// LS Electric XG5000 project: 과년71_1
// PLC NewPLC
// module base 0 slot 0: 입출력 모듈:XBC-DR20S (DC 24V 입력 12점, 릴레이 출력 8점)

PROGRAM NewProgram (task: 스캔 프로그램)

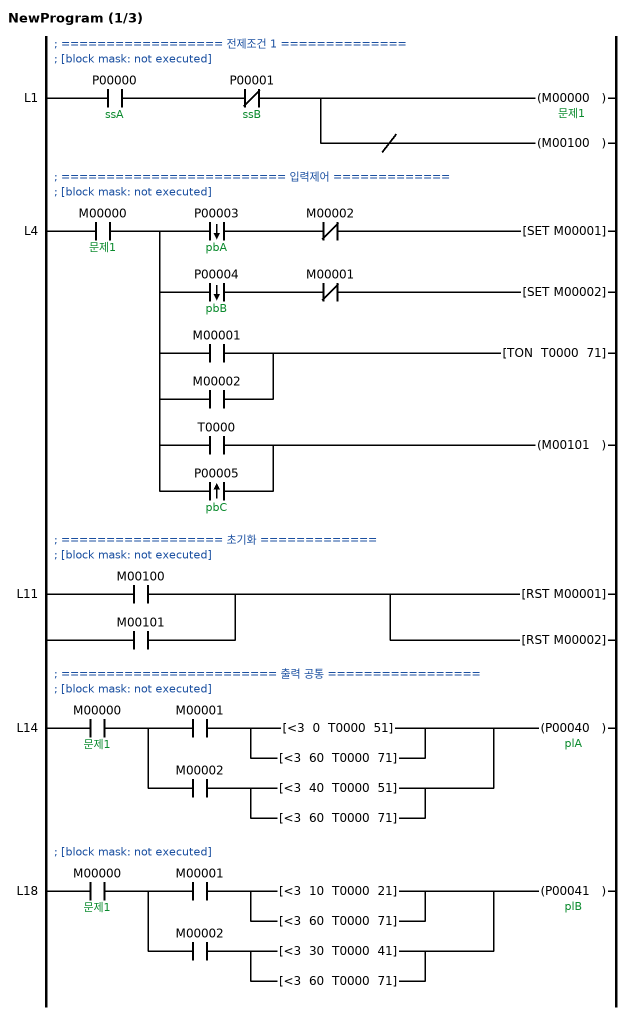
// ================== 전제조건 1 ==============
; L1 (block mask: not executed)
LOAD      P00000	// ssA
AND NOT   P00001	// ssB
OUT       M00000	// 문제1
NOT
OUT       M00100
// ========================= 입력제어 =============
; L4 (block mask: not executed)
LOAD      M00000	// 문제1
MPUSH
ANDN      P00003	// pbA
AND NOT   M00002
SET       M00001
MLOAD
ANDN      P00004	// pbB
AND NOT   M00001
SET       M00002
MLOAD
LOAD      M00001
OR        M00002
AND LOAD
TON       T0000 71
MPOP
LOAD      T0000
ORP       P00005	// pbC
AND LOAD
OUT       M00101
// ================== 초기화 =============
; L11 (block mask: not executed)
LOAD      M00100
OR        M00101
RST       M00001
RST       M00002
// ======================== 출력 공통 =================
; L14 (block mask: not executed)
LOAD      M00000	// 문제1
LOAD      M00001
LOAD<3    0 T0000 51
OR<3      60 T0000 71
AND LOAD
LOAD      M00002
LOAD<3    40 T0000 51
OR<3      60 T0000 71
AND LOAD
OR LOAD
AND LOAD
OUT       P00040	// plA
; L18 (block mask: not executed)
LOAD      M00000	// 문제1
LOAD      M00001
LOAD<3    10 T0000 21
OR<3      60 T0000 71
AND LOAD
LOAD      M00002
LOAD<3    30 T0000 41
OR<3      60 T0000 71
AND LOAD
OR LOAD
AND LOAD
OUT       P00041	// plB

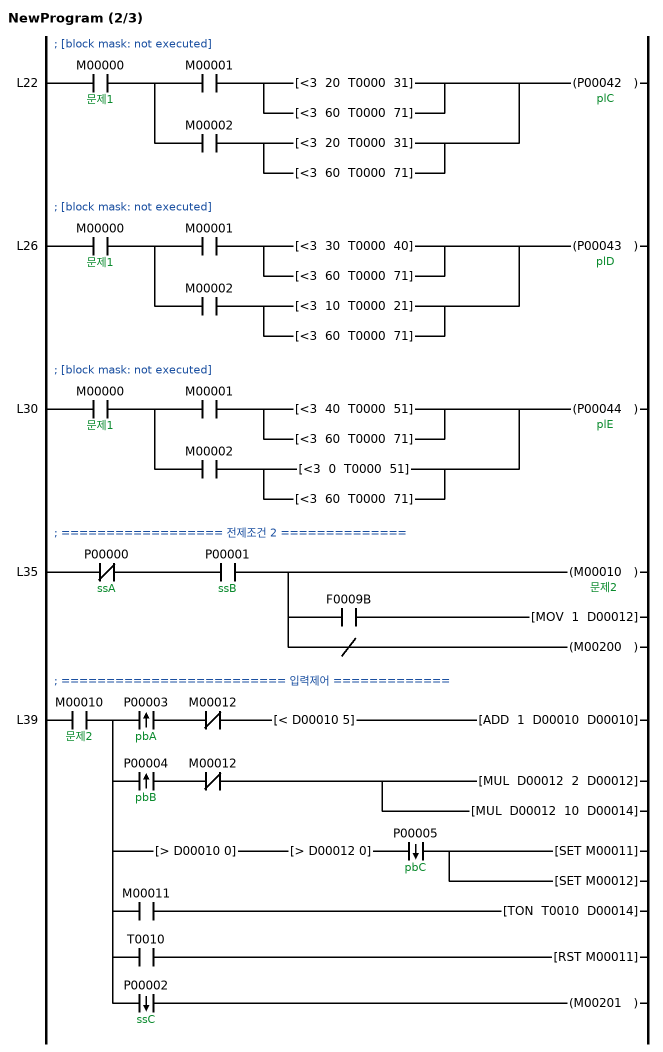
; L22 (block mask: not executed)
LOAD      M00000	// 문제1
LOAD      M00001
LOAD<3    20 T0000 31
OR<3      60 T0000 71
AND LOAD
LOAD      M00002
LOAD<3    20 T0000 31
OR<3      60 T0000 71
AND LOAD
OR LOAD
AND LOAD
OUT       P00042	// plC
; L26 (block mask: not executed)
LOAD      M00000	// 문제1
LOAD      M00001
LOAD<3    30 T0000 40
OR<3      60 T0000 71
AND LOAD
LOAD      M00002
LOAD<3    10 T0000 21
OR<3      60 T0000 71
AND LOAD
OR LOAD
AND LOAD
OUT       P00043	// plD
; L30 (block mask: not executed)
LOAD      M00000	// 문제1
LOAD      M00001
LOAD<3    40 T0000 51
OR<3      60 T0000 71
AND LOAD
LOAD      M00002
LOAD<3    0 T0000 51
OR<3      60 T0000 71
AND LOAD
OR LOAD
AND LOAD
OUT       P00044	// plE
// ================== 전제조건 2 ==============
; L35
LOAD NOT  P00000	// ssA
AND       P00001	// ssB
OUT       M00010	// 문제2
MPUSH
AND       F0009B
MOV       1 D00012
MPOP
NOT
OUT       M00200
// ========================= 입력제어 =============
; L39
LOAD      M00010	// 문제2
MPUSH
ANDP      P00003	// pbA
AND NOT   M00012
AND<      D00010 5
ADD       1 D00010 D00010
MLOAD
ANDP      P00004	// pbB
AND NOT   M00012
MUL       D00012 2 D00012
MUL       D00012 10 D00014
MLOAD
AND>      D00010 0
AND>      D00012 0
ANDN      P00005	// pbC
SET       M00011
SET       M00012
MLOAD
AND       M00011
TON       T0010 D00014
MLOAD
AND       T0010
RST       M00011
MPOP
ANDN      P00002	// ssC
OUT       M00201

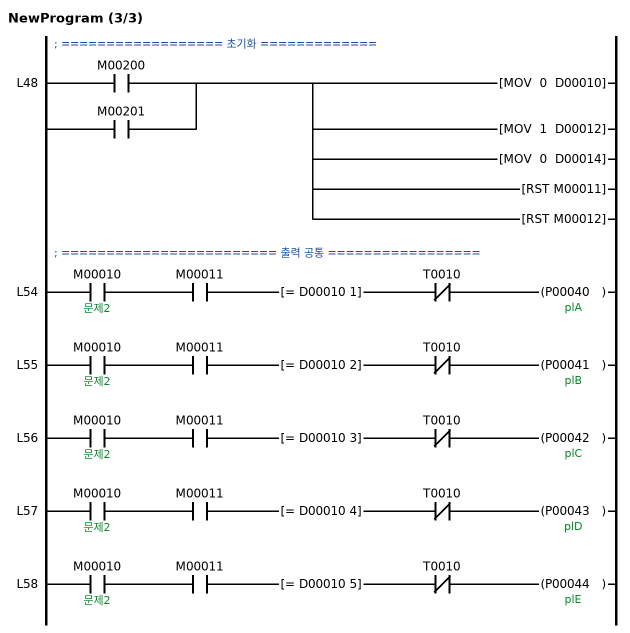
// ================== 초기화 =============
; L48
LOAD      M00200
OR        M00201
MOV       0 D00010
MOV       1 D00012
MOV       0 D00014
RST       M00011
RST       M00012
// ======================== 출력 공통 =================
; L54
LOAD      M00010	// 문제2
AND       M00011
AND=      D00010 1
AND NOT   T0010
OUT       P00040	// plA
; L55
LOAD      M00010	// 문제2
AND       M00011
AND=      D00010 2
AND NOT   T0010
OUT       P00041	// plB
; L56
LOAD      M00010	// 문제2
AND       M00011
AND=      D00010 3
AND NOT   T0010
OUT       P00042	// plC
; L57
LOAD      M00010	// 문제2
AND       M00011
AND=      D00010 4
AND NOT   T0010
OUT       P00043	// plD
; L58
LOAD      M00010	// 문제2
AND       M00011
AND=      D00010 5
AND NOT   T0010
OUT       P00044	// plE